Fanuc KAREL source: ka00118.KL

PROGRAM KA00118
%STACKSIZE=65535
%PRIORITY=65535
%NOLOCKGROUP
-- UNRESOLVED DECLARATIONS (source type spelling not recovered)
-- SRC : TYPE_0x001C (type_u16=0x001C)
-- DST : TYPE_0x001C (type_u16=0x001C)
BEGIN
-- UNRESOLVED_PC line 7 opcodes [9D 22 A5] marker_code=0
DST=SRC
END KA00118
